INTERFACE I_FallibleINT EXTENDS I_Fallible

PROPERTY Val : INT
GET
END_GET
END_PROPERTY

END_INTERFACE

(* stored: Version 1.1.0.1
   Itf I_FallibleINT: Id {9aed38e0-684d-430f-a26a-a236f4e39527}
   Property Val: Id {86952b0e-9d30-4a56-89f3-07afe624326d}
   Get Get: Id {ccc13ada-480b-4804-9ff5-c11adbb234ef} *)
